SYSTEM FestoMPS
  (* Version 1.0, Author, 4DIAC-Consortium *)
  APPLICATION PicknPlace
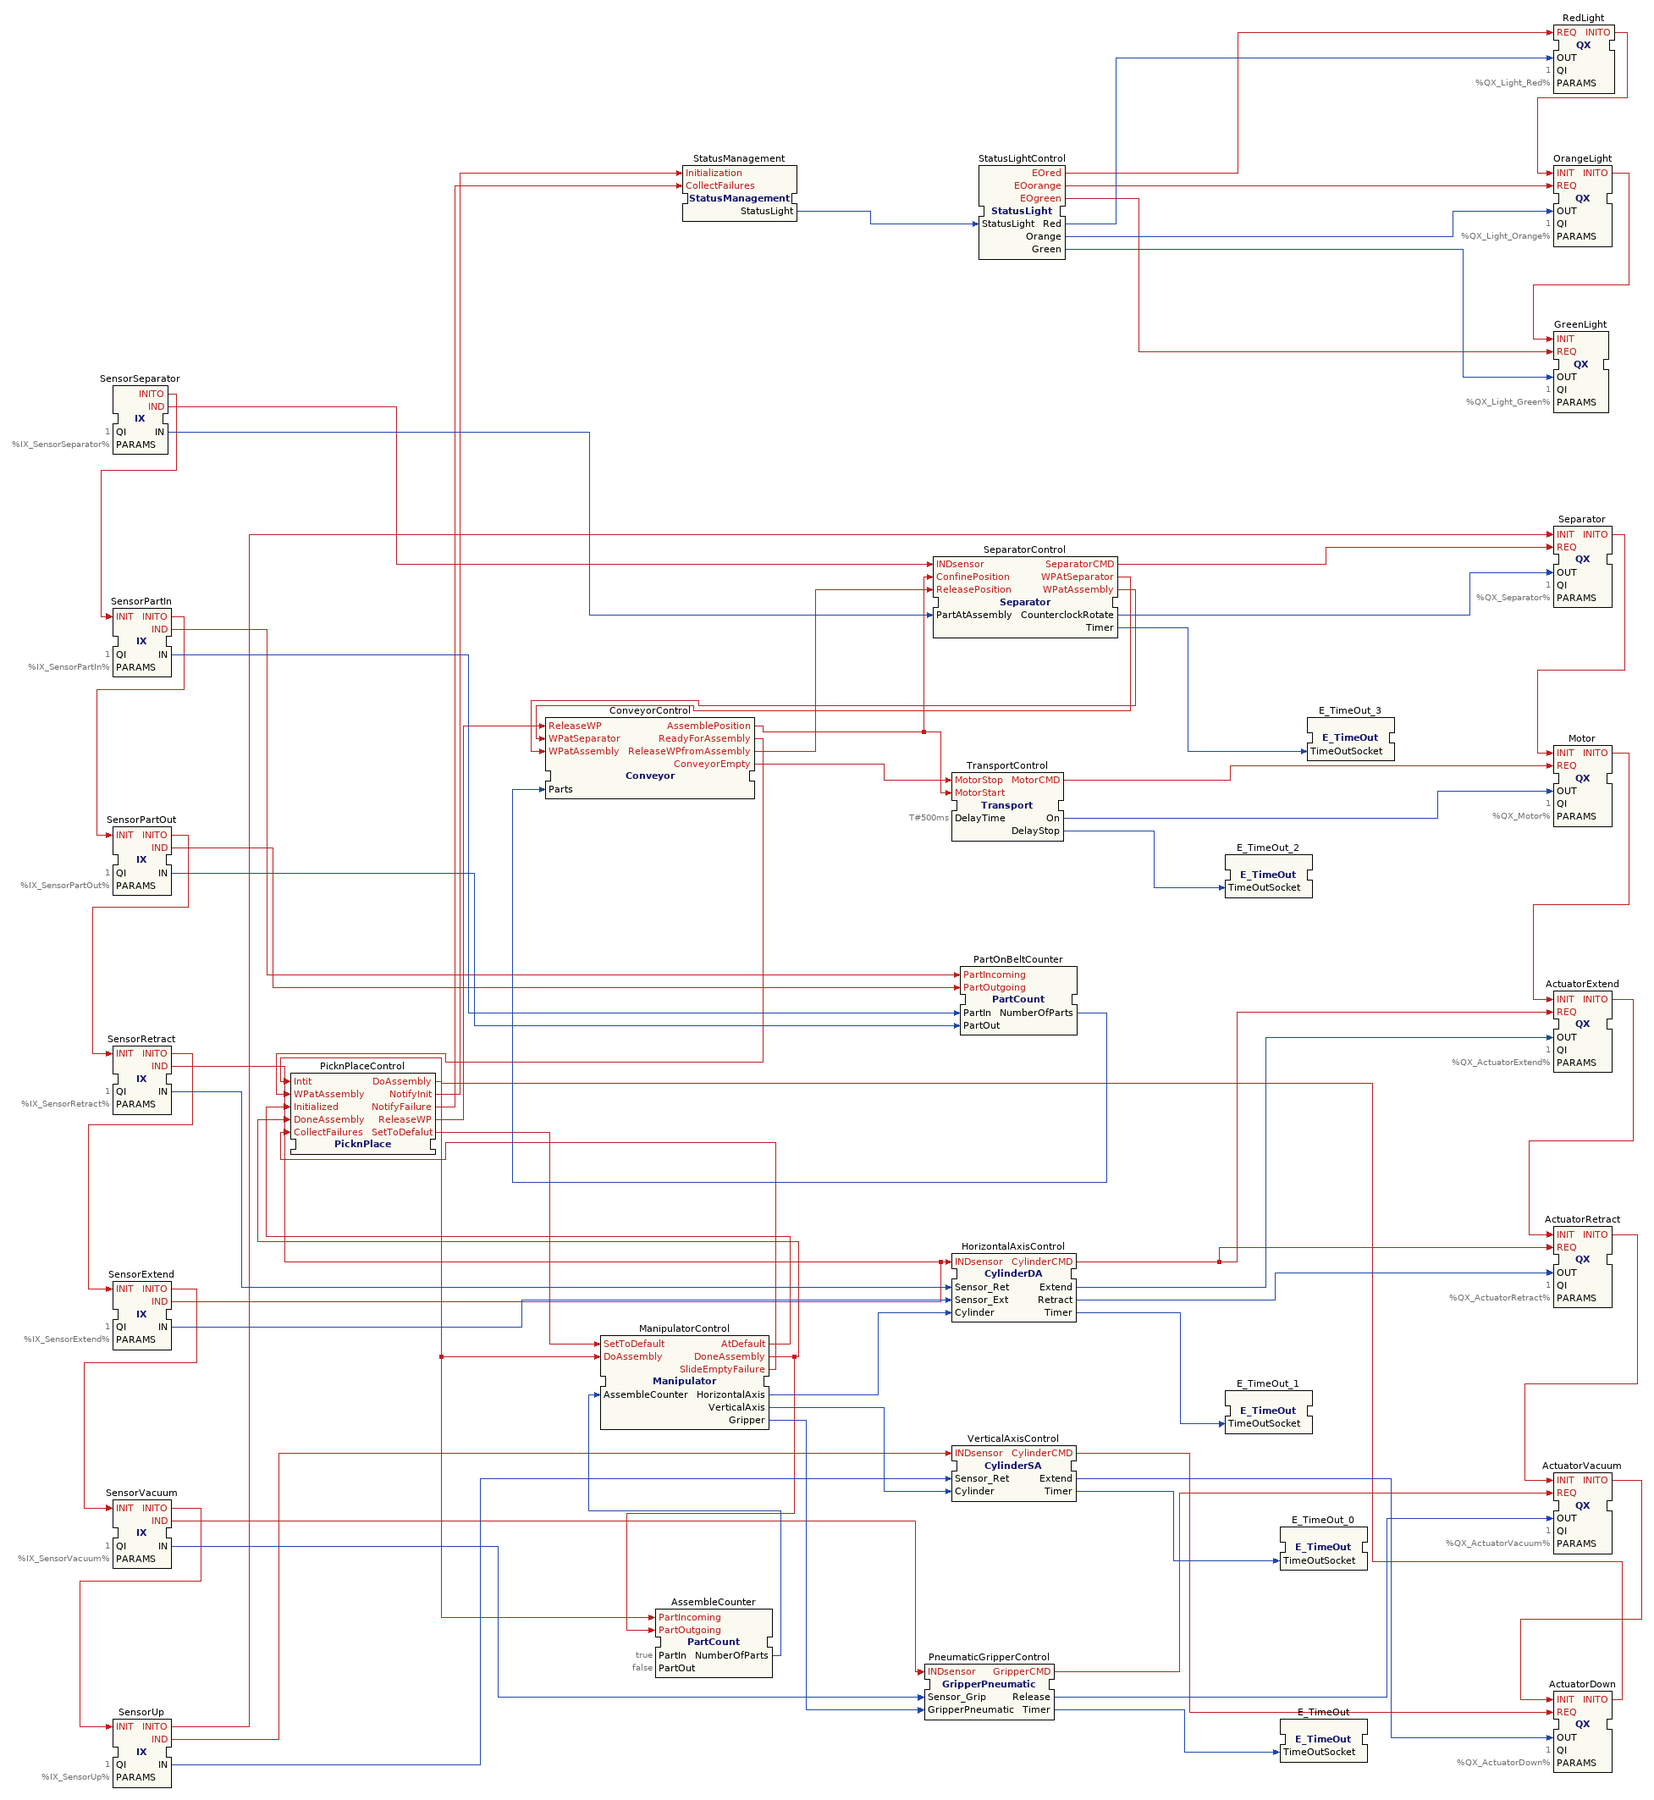
    FBS
      Motor : QX(QI := 1, PARAMS := %QX_Motor%);
      Separator : QX(QI := 1, PARAMS := %QX_Separator%);
      ActuatorDown : QX(QI := 1, PARAMS := %QX_ActuatorDown%);
      ActuatorVacuum : QX(QI := 1, PARAMS := %QX_ActuatorVacuum%);
      ActuatorRetract : QX(QI := 1, PARAMS := %QX_ActuatorRetract%);
      ActuatorExtend : QX(QI := 1, PARAMS := %QX_ActuatorExtend%);
      E_TimeOut : E_TimeOut;
      E_TimeOut_0 : E_TimeOut;
      E_TimeOut_1 : E_TimeOut;
      SensorSeparator : IX(QI := 1, PARAMS := %IX_SensorSeparator%);
      SensorPartIn : IX(QI := 1, PARAMS := %IX_SensorPartIn%);
      SensorPartOut : IX(QI := 1, PARAMS := %IX_SensorPartOut%);
      SensorRetract : IX(QI := 1, PARAMS := %IX_SensorRetract%);
      SensorVacuum : IX(QI := 1, PARAMS := %IX_SensorVacuum%);
      SensorExtend : IX(QI := 1, PARAMS := %IX_SensorExtend%);
      SensorUp : IX(QI := 1, PARAMS := %IX_SensorUp%);
      E_TimeOut_2 : E_TimeOut;
      GreenLight : QX(QI := 1, PARAMS := %QX_Light_Green%);
      RedLight : QX(QI := 1, PARAMS := %QX_Light_Red%);
      OrangeLight : QX(QI := 1, PARAMS := %QX_Light_Orange%);
      E_TimeOut_3 : E_TimeOut;
      PartOnBeltCounter : PartCount;
      AssembleCounter : PartCount(PartIn := true, PartOut := false);
      VerticalAxisControl : CylinderSA;
      PneumaticGripperControl : GripperPneumatic;
      HorizontalAxisControl : CylinderDA;
      PicknPlaceControl : PicknPlace;
      TransportControl : Transport(DelayTime := T#500ms);
      StatusLightControl : StatusLight;
      StatusManagement : StatusManagement;
      SeparatorControl : Separator;
      ConveyorControl : Conveyor;
      ManipulatorControl : Manipulator;
    END_FBS
    EVENT_CONNECTIONS
      Separator.INITO TO Motor.INIT;
      Motor.INITO TO ActuatorExtend.INIT;
      ActuatorExtend.INITO TO ActuatorRetract.INIT;
      ActuatorRetract.INITO TO ActuatorVacuum.INIT;
      ActuatorVacuum.INITO TO ActuatorDown.INIT;
      SensorSeparator.INITO TO SensorPartIn.INIT;
      SensorPartIn.INITO TO SensorPartOut.INIT;
      SensorPartOut.INITO TO SensorRetract.INIT;
      SensorRetract.INITO TO SensorExtend.INIT;
      SensorExtend.INITO TO SensorVacuum.INIT;
      SensorVacuum.INITO TO SensorUp.INIT;
      SensorUp.INITO TO Separator.INIT;
      RedLight.INITO TO OrangeLight.INIT;
      OrangeLight.INITO TO GreenLight.INIT;
      SensorPartIn.IND TO PartOnBeltCounter.PartIncoming;
      SensorPartOut.IND TO PartOnBeltCounter.PartOutgoing;
      SensorUp.IND TO VerticalAxisControl.INDsensor;
      VerticalAxisControl.CylinderCMD TO ActuatorDown.REQ;
      SensorVacuum.IND TO PneumaticGripperControl.INDsensor;
      PneumaticGripperControl.GripperCMD TO ActuatorVacuum.REQ;
      SensorRetract.IND TO HorizontalAxisControl.INDsensor;
      SensorExtend.IND TO HorizontalAxisControl.INDsensor;
      HorizontalAxisControl.CylinderCMD TO ActuatorRetract.REQ;
      ActuatorDown.INITO TO PicknPlaceControl.Intit;
      PicknPlaceControl.DoAssembly TO AssembleCounter.PartIncoming;
      HorizontalAxisControl.CylinderCMD TO ActuatorExtend.REQ;
      TransportControl.MotorCMD TO Motor.REQ;
      StatusLightControl.EOred TO RedLight.REQ;
      StatusLightControl.EOorange TO OrangeLight.REQ;
      StatusLightControl.EOgreen TO GreenLight.REQ;
      PicknPlaceControl.NotifyInit TO StatusManagement.Initialization;
      PicknPlaceControl.NotifyFailure TO StatusManagement.CollectFailures;
      SensorSeparator.IND TO SeparatorControl.INDsensor;
      SeparatorControl.SeparatorCMD TO Separator.REQ;
      PicknPlaceControl.ReleaseWP TO ConveyorControl.ReleaseWP;
      SeparatorControl.WPAtSeparator TO ConveyorControl.WPatSeparator;
      SeparatorControl.WPatAssembly TO ConveyorControl.WPatAssembly;
      ConveyorControl.AssemblePosition TO SeparatorControl.ConfinePosition;
      ConveyorControl.ReadyForAssembly TO PicknPlaceControl.WPatAssembly;
      ConveyorControl.ReleaseWPfromAssembly TO SeparatorControl.ReleasePosition;
      ConveyorControl.ConveyorEmpty TO TransportControl.MotorStop;
      ConveyorControl.AssemblePosition TO TransportControl.MotorStart;
      PicknPlaceControl.SetToDefalut TO ManipulatorControl.SetToDefault;
      PicknPlaceControl.DoAssembly TO ManipulatorControl.DoAssembly;
      ManipulatorControl.AtDefault TO PicknPlaceControl.Initialized;
      ManipulatorControl.DoneAssembly TO AssembleCounter.PartOutgoing;
      ManipulatorControl.DoneAssembly TO PicknPlaceControl.DoneAssembly;
      ManipulatorControl.SlideEmptyFailure TO PicknPlaceControl.CollectFailures;
    END_CONNECTIONS
    DATA_CONNECTIONS
      SensorPartIn.IN TO PartOnBeltCounter.PartIn;
      SensorPartOut.IN TO PartOnBeltCounter.PartOut;
      SensorUp.IN TO VerticalAxisControl.Sensor_Ret;
      VerticalAxisControl.Extend TO ActuatorDown.OUT;
      VerticalAxisControl.Timer TO E_TimeOut_0.TimeOutSocket;
      SensorVacuum.IN TO PneumaticGripperControl.Sensor_Grip;
      PneumaticGripperControl.Release TO ActuatorVacuum.OUT;
      PneumaticGripperControl.Timer TO E_TimeOut.TimeOutSocket;
      SensorRetract.IN TO HorizontalAxisControl.Sensor_Ret;
      SensorExtend.IN TO HorizontalAxisControl.Sensor_Ext;
      HorizontalAxisControl.Extend TO ActuatorExtend.OUT;
      HorizontalAxisControl.Retract TO ActuatorRetract.OUT;
      HorizontalAxisControl.Timer TO E_TimeOut_1.TimeOutSocket;
      TransportControl.On TO Motor.OUT;
      TransportControl.DelayStop TO E_TimeOut_2.TimeOutSocket;
      StatusLightControl.Red TO RedLight.OUT;
      StatusLightControl.Orange TO OrangeLight.OUT;
      StatusLightControl.Green TO GreenLight.OUT;
      StatusManagement.StatusLight TO StatusLightControl.StatusLight;
      SeparatorControl.CounterclockRotate TO Separator.OUT;
      SeparatorControl.Timer TO E_TimeOut_3.TimeOutSocket;
      SensorSeparator.IN TO SeparatorControl.PartAtAssembly;
      PartOnBeltCounter.NumberOfParts TO ConveyorControl.Parts;
      AssembleCounter.NumberOfParts TO ManipulatorControl.AssembleCounter;
      ManipulatorControl.HorizontalAxis TO HorizontalAxisControl.Cylinder;
      ManipulatorControl.VerticalAxis TO VerticalAxisControl.Cylinder;
      ManipulatorControl.Gripper TO PneumaticGripperControl.GripperPneumatic;
    END_CONNECTIONS
  END_APPLICATION
  DEVICE PicknPlaceStatus : GenericFORTE(MGR_ID := %PicknPlaceStatusController%:61499)
    RESOURCE FORTE : EMB_RES
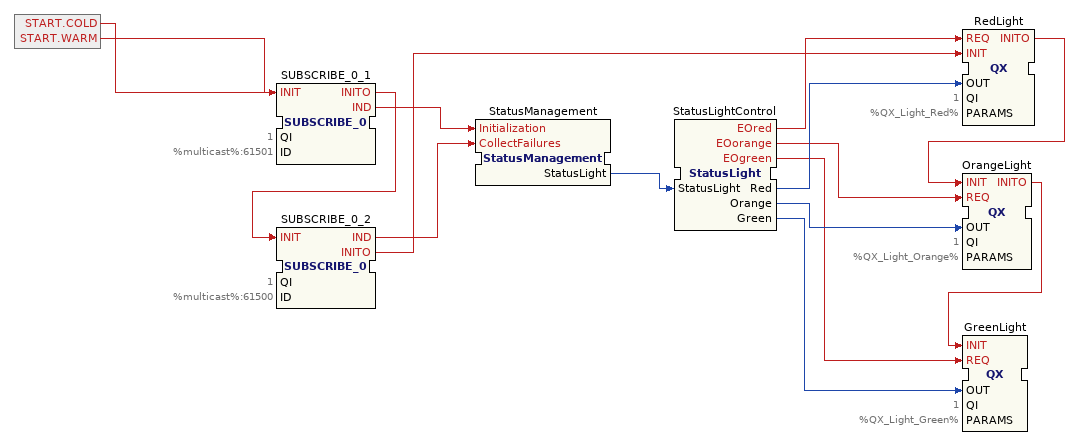
      FBS
        SUBSCRIBE_0_1 : SUBSCRIBE_0(QI := 1, ID := %multicast%:61501);
        SUBSCRIBE_0_2 : SUBSCRIBE_0(QI := 1, ID := %multicast%:61500);
        StatusManagement : StatusManagement;
        StatusLightControl : StatusLight;
        RedLight : QX(QI := 1, PARAMS := %QX_Light_Red%);
        OrangeLight : QX(QI := 1, PARAMS := %QX_Light_Orange%);
        GreenLight : QX(QI := 1, PARAMS := %QX_Light_Green%);
      END_FBS
      EVENT_CONNECTIONS
        START.COLD TO SUBSCRIBE_0_1.INIT;
        SUBSCRIBE_0_1.INITO TO SUBSCRIBE_0_2.INIT;
        StatusLightControl.EOred TO RedLight.REQ;
        RedLight.INITO TO OrangeLight.INIT;
        StatusLightControl.EOorange TO OrangeLight.REQ;
        OrangeLight.INITO TO GreenLight.INIT;
        StatusLightControl.EOgreen TO GreenLight.REQ;
        SUBSCRIBE_0_1.IND TO StatusManagement.Initialization;
        SUBSCRIBE_0_2.IND TO StatusManagement.CollectFailures;
        SUBSCRIBE_0_2.INITO TO RedLight.INIT;
        START.WARM TO SUBSCRIBE_0_1.INIT;
      END_CONNECTIONS
      DATA_CONNECTIONS
        StatusManagement.StatusLight TO StatusLightControl.StatusLight;
        StatusLightControl.Red TO RedLight.OUT;
        StatusLightControl.Orange TO OrangeLight.OUT;
        StatusLightControl.Green TO GreenLight.OUT;
      END_CONNECTIONS
    END_RESOURCE
  END_DEVICE
  DEVICE PicknPlace : GenericFORTE(MGR_ID := %PicknPlaceController%:61499)
    RESOURCE FORTE : EMB_RES
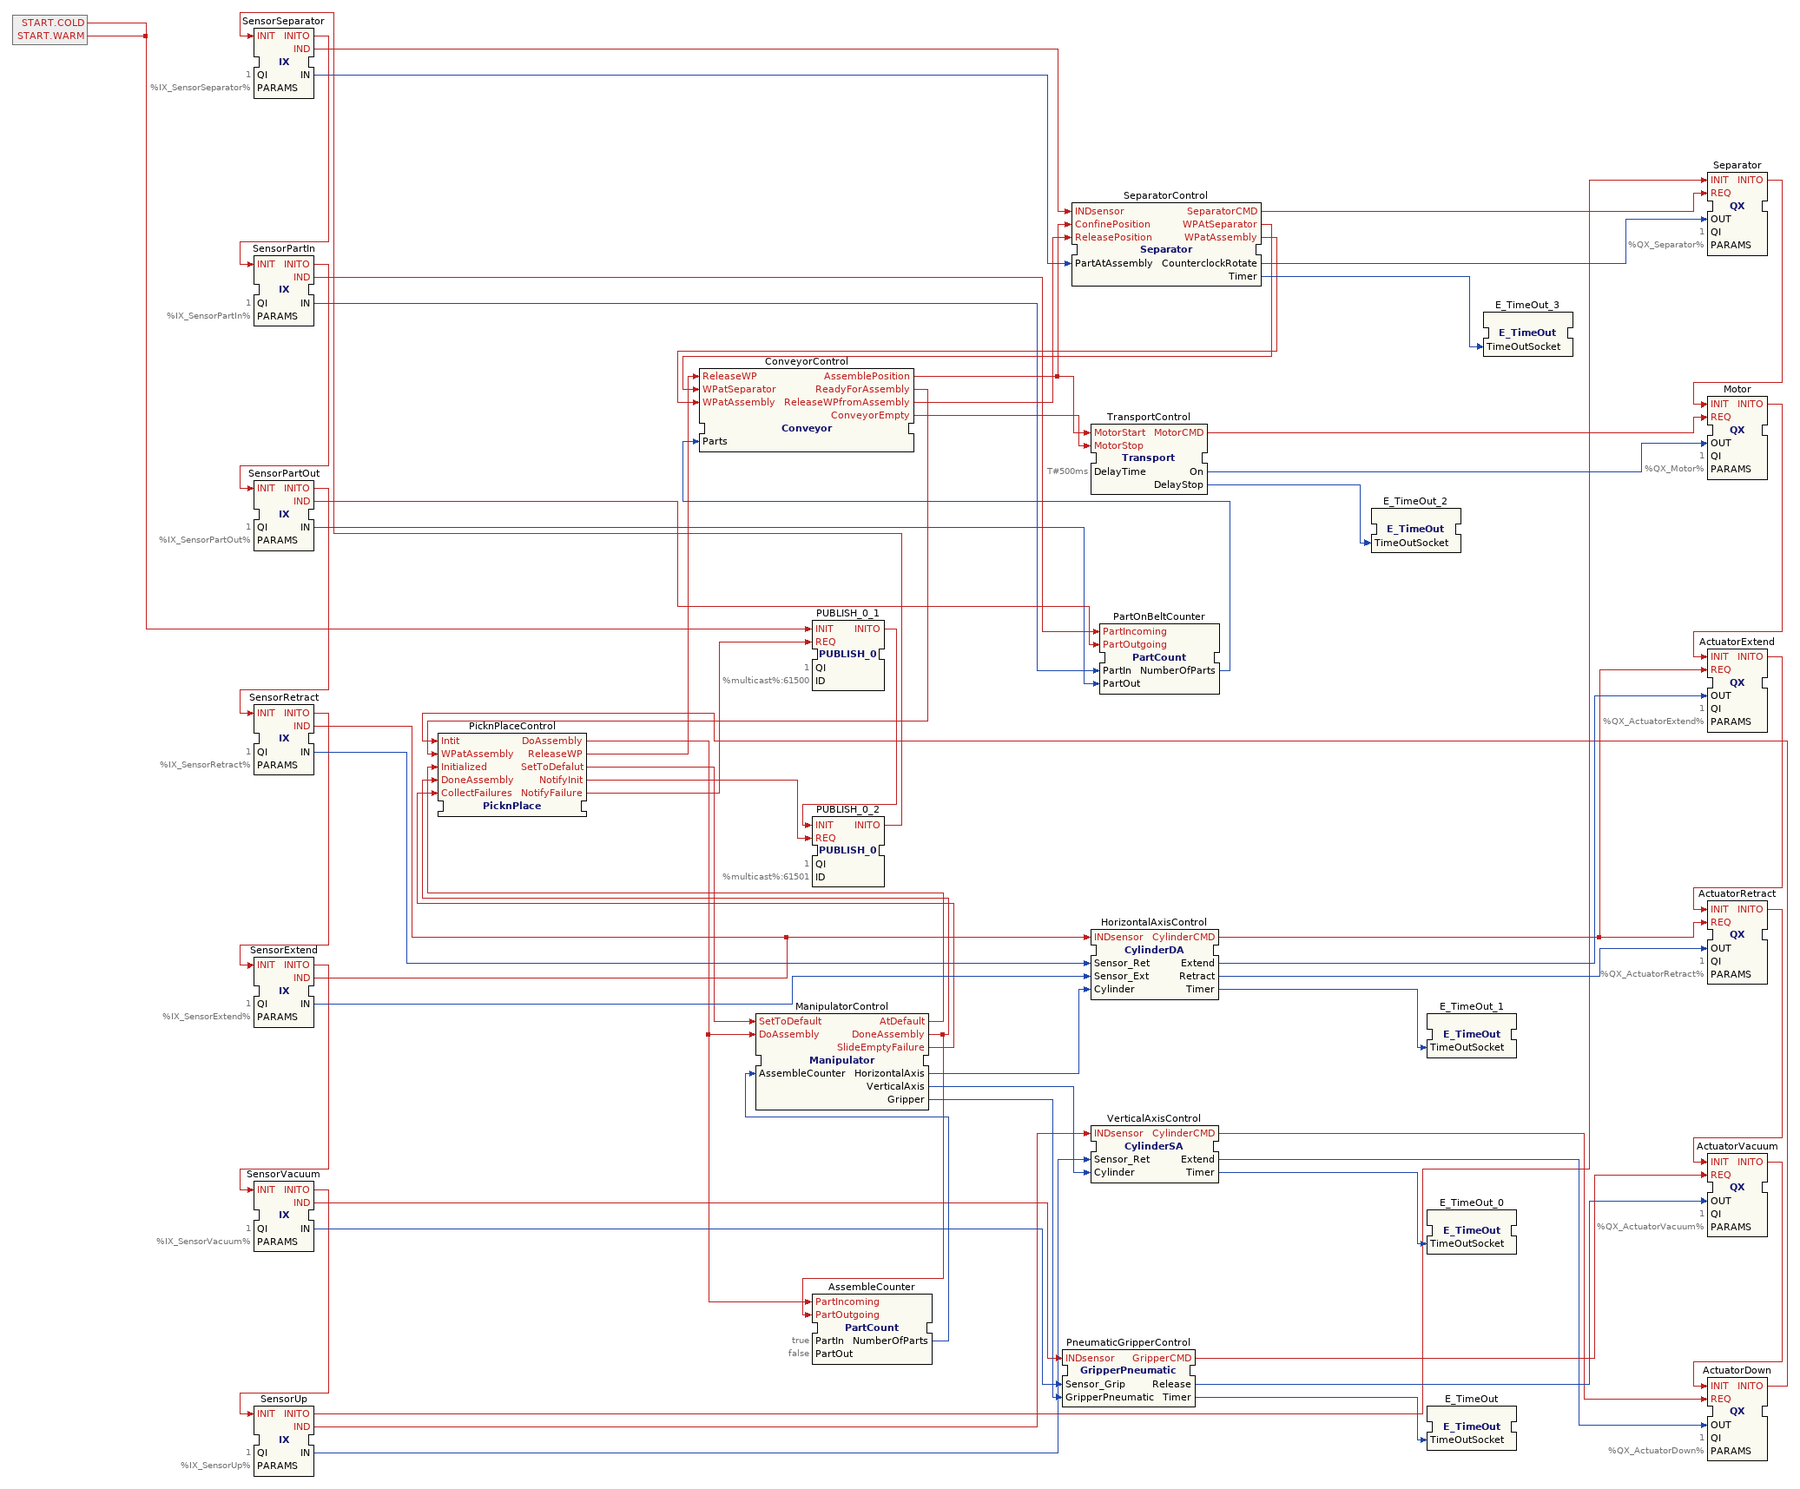
      FBS
        PUBLISH_0_1 : PUBLISH_0(QI := 1, ID := %multicast%:61500);
        PUBLISH_0_2 : PUBLISH_0(QI := 1, ID := %multicast%:61501);
        Motor : QX(QI := 1, PARAMS := %QX_Motor%);
        Separator : QX(QI := 1, PARAMS := %QX_Separator%);
        ActuatorDown : QX(QI := 1, PARAMS := %QX_ActuatorDown%);
        ActuatorVacuum : QX(QI := 1, PARAMS := %QX_ActuatorVacuum%);
        ActuatorRetract : QX(QI := 1, PARAMS := %QX_ActuatorRetract%);
        ActuatorExtend : QX(QI := 1, PARAMS := %QX_ActuatorExtend%);
        E_TimeOut : E_TimeOut;
        E_TimeOut_0 : E_TimeOut;
        E_TimeOut_1 : E_TimeOut;
        SensorSeparator : IX(QI := 1, PARAMS := %IX_SensorSeparator%);
        SensorPartIn : IX(QI := 1, PARAMS := %IX_SensorPartIn%);
        SensorPartOut : IX(QI := 1, PARAMS := %IX_SensorPartOut%);
        SensorRetract : IX(QI := 1, PARAMS := %IX_SensorRetract%);
        SensorVacuum : IX(QI := 1, PARAMS := %IX_SensorVacuum%);
        SensorExtend : IX(QI := 1, PARAMS := %IX_SensorExtend%);
        SensorUp : IX(QI := 1, PARAMS := %IX_SensorUp%);
        E_TimeOut_2 : E_TimeOut;
        E_TimeOut_3 : E_TimeOut;
        PartOnBeltCounter : PartCount;
        AssembleCounter : PartCount(PartIn := true, PartOut := false);
        VerticalAxisControl : CylinderSA;
        PneumaticGripperControl : GripperPneumatic;
        HorizontalAxisControl : CylinderDA;
        PicknPlaceControl : PicknPlace;
        TransportControl : Transport(DelayTime := T#500ms);
        SeparatorControl : Separator;
        ConveyorControl : Conveyor;
        ManipulatorControl : Manipulator;
      END_FBS
      EVENT_CONNECTIONS
        PUBLISH_0_1.INITO TO PUBLISH_0_2.INIT;
        START.COLD TO PUBLISH_0_1.INIT;
        START.WARM TO PUBLISH_0_1.INIT;
        Separator.INITO TO Motor.INIT;
        ActuatorVacuum.INITO TO ActuatorDown.INIT;
        ActuatorRetract.INITO TO ActuatorVacuum.INIT;
        Motor.INITO TO ActuatorExtend.INIT;
        ActuatorExtend.INITO TO ActuatorRetract.INIT;
        SensorSeparator.INITO TO SensorPartIn.INIT;
        SensorPartIn.INITO TO SensorPartOut.INIT;
        SensorPartOut.INITO TO SensorRetract.INIT;
        SensorRetract.INITO TO SensorExtend.INIT;
        SensorExtend.INITO TO SensorVacuum.INIT;
        SensorVacuum.INITO TO SensorUp.INIT;
        SensorUp.INITO TO Separator.INIT;
        SensorPartIn.IND TO PartOnBeltCounter.PartIncoming;
        SensorPartOut.IND TO PartOnBeltCounter.PartOutgoing;
        SensorUp.IND TO VerticalAxisControl.INDsensor;
        VerticalAxisControl.CylinderCMD TO ActuatorDown.REQ;
        SensorVacuum.IND TO PneumaticGripperControl.INDsensor;
        PneumaticGripperControl.GripperCMD TO ActuatorVacuum.REQ;
        SensorRetract.IND TO HorizontalAxisControl.INDsensor;
        SensorExtend.IND TO HorizontalAxisControl.INDsensor;
        HorizontalAxisControl.CylinderCMD TO ActuatorRetract.REQ;
        HorizontalAxisControl.CylinderCMD TO ActuatorExtend.REQ;
        ActuatorDown.INITO TO PicknPlaceControl.Intit;
        PicknPlaceControl.DoAssembly TO AssembleCounter.PartIncoming;
        TransportControl.MotorCMD TO Motor.REQ;
        SensorSeparator.IND TO SeparatorControl.INDsensor;
        SeparatorControl.SeparatorCMD TO Separator.REQ;
        PicknPlaceControl.ReleaseWP TO ConveyorControl.ReleaseWP;
        SeparatorControl.WPAtSeparator TO ConveyorControl.WPatSeparator;
        SeparatorControl.WPatAssembly TO ConveyorControl.WPatAssembly;
        ConveyorControl.AssemblePosition TO SeparatorControl.ConfinePosition;
        ConveyorControl.AssemblePosition TO TransportControl.MotorStart;
        ConveyorControl.ReadyForAssembly TO PicknPlaceControl.WPatAssembly;
        ConveyorControl.ReleaseWPfromAssembly TO SeparatorControl.ReleasePosition;
        ConveyorControl.ConveyorEmpty TO TransportControl.MotorStop;
        PicknPlaceControl.SetToDefalut TO ManipulatorControl.SetToDefault;
        PicknPlaceControl.DoAssembly TO ManipulatorControl.DoAssembly;
        ManipulatorControl.AtDefault TO PicknPlaceControl.Initialized;
        ManipulatorControl.DoneAssembly TO AssembleCounter.PartOutgoing;
        ManipulatorControl.DoneAssembly TO PicknPlaceControl.DoneAssembly;
        ManipulatorControl.SlideEmptyFailure TO PicknPlaceControl.CollectFailures;
        PicknPlaceControl.NotifyInit TO PUBLISH_0_2.REQ;
        PicknPlaceControl.NotifyFailure TO PUBLISH_0_1.REQ;
        PUBLISH_0_2.INITO TO SensorSeparator.INIT;
      END_CONNECTIONS
      DATA_CONNECTIONS
        SensorPartIn.IN TO PartOnBeltCounter.PartIn;
        SensorPartOut.IN TO PartOnBeltCounter.PartOut;
        SensorUp.IN TO VerticalAxisControl.Sensor_Ret;
        VerticalAxisControl.Extend TO ActuatorDown.OUT;
        VerticalAxisControl.Timer TO E_TimeOut_0.TimeOutSocket;
        SensorVacuum.IN TO PneumaticGripperControl.Sensor_Grip;
        PneumaticGripperControl.Release TO ActuatorVacuum.OUT;
        PneumaticGripperControl.Timer TO E_TimeOut.TimeOutSocket;
        SensorRetract.IN TO HorizontalAxisControl.Sensor_Ret;
        SensorExtend.IN TO HorizontalAxisControl.Sensor_Ext;
        HorizontalAxisControl.Extend TO ActuatorExtend.OUT;
        HorizontalAxisControl.Retract TO ActuatorRetract.OUT;
        HorizontalAxisControl.Timer TO E_TimeOut_1.TimeOutSocket;
        TransportControl.On TO Motor.OUT;
        TransportControl.DelayStop TO E_TimeOut_2.TimeOutSocket;
        SensorSeparator.IN TO SeparatorControl.PartAtAssembly;
        SeparatorControl.CounterclockRotate TO Separator.OUT;
        SeparatorControl.Timer TO E_TimeOut_3.TimeOutSocket;
        PartOnBeltCounter.NumberOfParts TO ConveyorControl.Parts;
        AssembleCounter.NumberOfParts TO ManipulatorControl.AssembleCounter;
        ManipulatorControl.HorizontalAxis TO HorizontalAxisControl.Cylinder;
        ManipulatorControl.VerticalAxis TO VerticalAxisControl.Cylinder;
        ManipulatorControl.Gripper TO PneumaticGripperControl.GripperPneumatic;
      END_CONNECTIONS
    END_RESOURCE
  END_DEVICE
  MAPPINGS
    PicknPlace.Motor ON PicknPlace.FORTE.Motor;
    PicknPlace.Separator ON PicknPlace.FORTE.Separator;
    PicknPlace.ActuatorDown ON PicknPlace.FORTE.ActuatorDown;
    PicknPlace.ActuatorVacuum ON PicknPlace.FORTE.ActuatorVacuum;
    PicknPlace.ActuatorRetract ON PicknPlace.FORTE.ActuatorRetract;
    PicknPlace.ActuatorExtend ON PicknPlace.FORTE.ActuatorExtend;
    PicknPlace.E_TimeOut ON PicknPlace.FORTE.E_TimeOut;
    PicknPlace.E_TimeOut_0 ON PicknPlace.FORTE.E_TimeOut_0;
    PicknPlace.E_TimeOut_1 ON PicknPlace.FORTE.E_TimeOut_1;
    PicknPlace.SensorSeparator ON PicknPlace.FORTE.SensorSeparator;
    PicknPlace.SensorPartIn ON PicknPlace.FORTE.SensorPartIn;
    PicknPlace.SensorPartOut ON PicknPlace.FORTE.SensorPartOut;
    PicknPlace.SensorRetract ON PicknPlace.FORTE.SensorRetract;
    PicknPlace.SensorVacuum ON PicknPlace.FORTE.SensorVacuum;
    PicknPlace.SensorExtend ON PicknPlace.FORTE.SensorExtend;
    PicknPlace.SensorUp ON PicknPlace.FORTE.SensorUp;
    PicknPlace.E_TimeOut_2 ON PicknPlace.FORTE.E_TimeOut_2;
    PicknPlace.GreenLight ON PicknPlaceStatus.FORTE.GreenLight;
    PicknPlace.RedLight ON PicknPlaceStatus.FORTE.RedLight;
    PicknPlace.OrangeLight ON PicknPlaceStatus.FORTE.OrangeLight;
    PicknPlace.E_TimeOut_3 ON PicknPlace.FORTE.E_TimeOut_3;
    PicknPlace.PartOnBeltCounter ON PicknPlace.FORTE.PartOnBeltCounter;
    PicknPlace.AssembleCounter ON PicknPlace.FORTE.AssembleCounter;
    PicknPlace.VerticalAxisControl ON PicknPlace.FORTE.VerticalAxisControl;
    PicknPlace.PneumaticGripperControl ON PicknPlace.FORTE.PneumaticGripperControl;
    PicknPlace.HorizontalAxisControl ON PicknPlace.FORTE.HorizontalAxisControl;
    PicknPlace.PicknPlaceControl ON PicknPlace.FORTE.PicknPlaceControl;
    PicknPlace.TransportControl ON PicknPlace.FORTE.TransportControl;
    PicknPlace.StatusLightControl ON PicknPlaceStatus.FORTE.StatusLightControl;
    PicknPlace.StatusManagement ON PicknPlaceStatus.FORTE.StatusManagement;
    PicknPlace.SeparatorControl ON PicknPlace.FORTE.SeparatorControl;
    PicknPlace.ConveyorControl ON PicknPlace.FORTE.ConveyorControl;
    PicknPlace.ManipulatorControl ON PicknPlace.FORTE.ManipulatorControl;
  END_MAPPINGS
  SEGMENTS
    Ethernet : Ethernet;
  END_SEGMENTS
  LINKS
    PicknPlaceStatus => Ethernet;
    PicknPlace => Ethernet;
  END_LINKS
END_SYSTEM
